(* CODESYS project ESCADA.project

Project tree, tasks and I/O mapping:
  Device : CODESYS Control Win V3, 3S - Smart Software Solutions GmbH, order no. 305021, version 3.5.11.30
    application Application
      libraries: Standard, * (System)
      task MainTask (cyclic, interval t#20ms, priority 1) calls PLC_PRG
      program PLC_PRG [LD]
*)

// Device/Application/PLC_PRG
PROGRAM PLC_PRG
VAR
	P1: BOOL;                       // SENSOR DE INICO DA ESCADA
	P2: BOOL;                       // SENSOR DE TOPO DA ESCADA
	AUX: BOOL;                      // AUXILIAR DO MOTOR
	S1: BOOL;                       // BOTAO RETENTIVO START/STOP
	KM: BOOL;                       // CONTATOR DO MOTOR
	TOF_1: TOF;
	ET1: TIME;
END_VAR
VAR // added by the converter: edge detectors and wires of the graphical bodies
    _ft1, _ft2, _ft3 : F_TRIG;
END_VAR

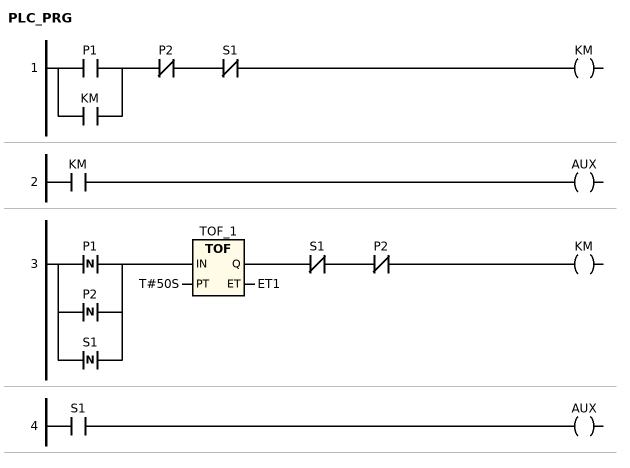
// NETWORK 1
KM := (P1 OR KM) AND NOT P2 AND NOT S1;

// NETWORK 2
AUX := KM;

// NETWORK 3
_ft1(CLK := P1);
_ft2(CLK := P2);
_ft3(CLK := S1);
TOF_1(IN := _ft1.Q OR _ft2.Q OR _ft3.Q, PT := T#50S, ET => ET1); // TOF
KM := TOF_1.Q AND NOT S1 AND NOT P2;

// NETWORK 4
AUX := S1;

END_PROGRAM
